TYPE ParallelUnitsStatus :
STRUCT
	PressureSupplyCSP: REAL; // Calculated Set Point for Master/Slave
	PressureExtractCSP: REAL; // Calculated Set Point for Master/Slave
	MasterActive: BOOL;
	IsMaster: BOOL;
	IsSlave: BOOL;
	SupplyFanSpeed: LREAL;
	ExtractFanSpeed: LREAL;
	IsRunning: BOOL;
	ResetAlarmMaster: BOOL;
	FireSupplyMaster: BOOL;
	FireExtractMaster: BOOL;
	FreezeMaster: BOOL;
	ResetAlarmSlave: BOOL;
	FireSupplySlave: BOOL;
	FireExtractSlave: BOOL;
	FreezeSlave: BOOL;
END_STRUCT
END_TYPE

(* stored: Version 1.1.0.1, ProductVersion 3.1.4024.6
   DUT ParallelUnitsStatus: Id {cc155ffc-f805-41ba-9ea5-38e44e17862e} *)
